// ---- POUs/Alle_Rum/Gange/Gang_5_153A/Visualization_4_330_1_1.TcVIS
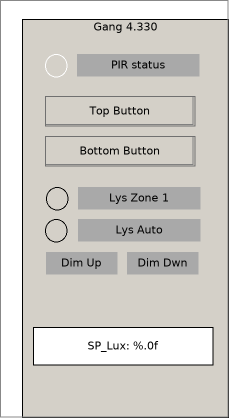
VISUALIZATION Visualization_4_330_1_1  // 229x418
    RoundedRectangle (22,19 207x399), "Gang 4.330"
    Rectangle (33,327 180x38), "SP_Lux: %.0f", text variable: P_Gang_5_135A.arrfbLysGruppe[1].fbLightCtrl.fLuxZone1
    Button (45,96 150x30), "Top Button"
        tap P_Gang_5_135A.bTopButtonZone1_Visu
    Button (45,136 150x30), "Bottom Button"
        tap P_Gang_5_135A.bBottomButtonZone1_Visu
    Ellipse (46,187 22x23), colour toggle: P_Gang_5_135A.fbLys.fbLightCtrl.bOnZone1
    Rectangle (78,187 122x22), "Lys Zone 1"
    Rectangle (46,252 71x22), "Dim Up", colour toggle: P_Gang_5_135A.arrfbLysGruppe[1].fbLightCtrl.bDimUp
    Rectangle (127,252 71x22), "Dim Dwn", colour toggle: P_Gang_5_135A.arrfbLysGruppe[1].fbLightCtrl.bDimDwn
    Ellipse (45,219 22x23), colour toggle: P_Gang_5_135A.arrfbLysGruppe[1].fbLightCtrl.bAutoZone1
    Rectangle (78,219 122x22), "Lys Auto"
    Ellipse (45,54 22x23), colour toggle: P_Gang_5_135A.arrfbLysGruppe[1].fbLightCtrl.bPIR
    Rectangle (77,54 122x22), "PIR status"
END_VISUALIZATION

// ---- POUs/Alle_Rum/Gange/Gang_5_149/Visualization_4_330_1_1_2.TcVIS
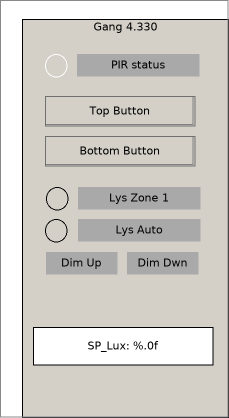
VISUALIZATION Visualization_4_330_1_1_2  // 229x418
    RoundedRectangle (22,19 207x399), "Gang 4.330"
    Rectangle (33,327 180x38), "SP_Lux: %.0f", text variable: P_Gang_5_135A.arrfbLysGruppe[1].fbLightCtrl.fLuxZone1
    Button (45,96 150x30), "Top Button"
        tap P_Gang_5_135A.bTopButtonZone1_Visu
    Button (45,136 150x30), "Bottom Button"
        tap P_Gang_5_135A.bBottomButtonZone1_Visu
    Ellipse (46,187 22x23), colour toggle: P_Gang_5_135A.fbLys.fbLightCtrl.bOnZone1
    Rectangle (78,187 122x22), "Lys Zone 1"
    Rectangle (46,252 71x22), "Dim Up", colour toggle: P_Gang_5_135A.arrfbLysGruppe[1].fbLightCtrl.bDimUp
    Rectangle (127,252 71x22), "Dim Dwn", colour toggle: P_Gang_5_135A.arrfbLysGruppe[1].fbLightCtrl.bDimDwn
    Ellipse (45,219 22x23), colour toggle: P_Gang_5_135A.arrfbLysGruppe[1].fbLightCtrl.bAutoZone1
    Rectangle (78,219 122x22), "Lys Auto"
    Ellipse (45,54 22x23), colour toggle: P_Gang_5_135A.arrfbLysGruppe[1].fbLightCtrl.bPIR
    Rectangle (77,54 122x22), "PIR status"
END_VISUALIZATION

// ---- POUs/Alle_Rum/Gange/Gang_7_119/Visualization_4_330_1_1_3.TcVIS
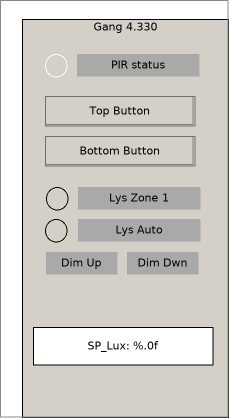
VISUALIZATION Visualization_4_330_1_1_3  // 229x418
    RoundedRectangle (22,19 207x399), "Gang 4.330"
    Rectangle (33,327 180x38), "SP_Lux: %.0f", text variable: P_Gang_5_135A.arrfbLysGruppe[1].fbLightCtrl.fLuxZone1
    Button (45,96 150x30), "Top Button"
        tap P_Gang_5_135A.bTopButtonZone1_Visu
    Button (45,136 150x30), "Bottom Button"
        tap P_Gang_5_135A.bBottomButtonZone1_Visu
    Ellipse (46,187 22x23), colour toggle: P_Gang_5_135A.fbLys.fbLightCtrl.bOnZone1
    Rectangle (78,187 122x22), "Lys Zone 1"
    Rectangle (46,252 71x22), "Dim Up", colour toggle: P_Gang_5_135A.arrfbLysGruppe[1].fbLightCtrl.bDimUp
    Rectangle (127,252 71x22), "Dim Dwn", colour toggle: P_Gang_5_135A.arrfbLysGruppe[1].fbLightCtrl.bDimDwn
    Ellipse (45,219 22x23), colour toggle: P_Gang_5_135A.arrfbLysGruppe[1].fbLightCtrl.bAutoZone1
    Rectangle (78,219 122x22), "Lys Auto"
    Ellipse (45,54 22x23), colour toggle: P_Gang_5_135A.arrfbLysGruppe[1].fbLightCtrl.bPIR
    Rectangle (77,54 122x22), "PIR status"
END_VISUALIZATION

// ---- POUs/Alle_Rum/Gange/Gang_5_153B/Visualization_4_330_1_1_1_1_1.TcVIS
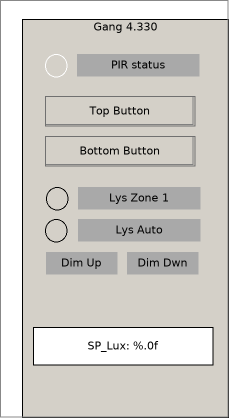
VISUALIZATION Visualization_4_330_1_1_1_1_1  // 229x418
    RoundedRectangle (22,19 207x399), "Gang 4.330"
    Rectangle (33,327 180x38), "SP_Lux: %.0f", text variable: P_Gang_5_135A.arrfbLysGruppe[1].fbLightCtrl.fLuxZone1
    Button (45,96 150x30), "Top Button"
        tap P_Gang_5_135A.bTopButtonZone1_Visu
    Button (45,136 150x30), "Bottom Button"
        tap P_Gang_5_135A.bBottomButtonZone1_Visu
    Ellipse (46,187 22x23), colour toggle: P_Gang_5_135A.fbLys.fbLightCtrl.bOnZone1
    Rectangle (78,187 122x22), "Lys Zone 1"
    Rectangle (46,252 71x22), "Dim Up", colour toggle: P_Gang_5_135A.arrfbLysGruppe[1].fbLightCtrl.bDimUp
    Rectangle (127,252 71x22), "Dim Dwn", colour toggle: P_Gang_5_135A.arrfbLysGruppe[1].fbLightCtrl.bDimDwn
    Ellipse (45,219 22x23), colour toggle: P_Gang_5_135A.arrfbLysGruppe[1].fbLightCtrl.bAutoZone1
    Rectangle (78,219 122x22), "Lys Auto"
    Ellipse (45,54 22x23), colour toggle: P_Gang_5_135A.arrfbLysGruppe[1].fbLightCtrl.bPIR
    Rectangle (77,54 122x22), "PIR status"
END_VISUALIZATION

// ---- POUs/Alle_Rum/Gange/Gang_5_145B/Visualization_4_330_1_1_1_1_1_1.TcVIS
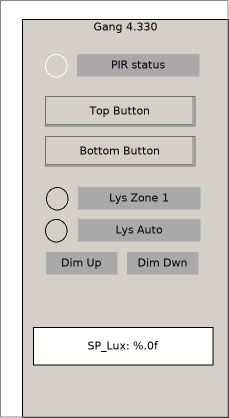
VISUALIZATION Visualization_4_330_1_1_1_1_1_1  // 229x418
    RoundedRectangle (22,19 207x399), "Gang 4.330"
    Rectangle (33,327 180x38), "SP_Lux: %.0f", text variable: P_Gang_5_135A.arrfbLysGruppe[1].fbLightCtrl.fLuxZone1
    Button (45,96 150x30), "Top Button"
        tap P_Gang_5_135A.bTopButtonZone1_Visu
    Button (45,136 150x30), "Bottom Button"
        tap P_Gang_5_135A.bBottomButtonZone1_Visu
    Ellipse (46,187 22x23), colour toggle: P_Gang_5_135A.fbLys.fbLightCtrl.bOnZone1
    Rectangle (78,187 122x22), "Lys Zone 1"
    Rectangle (46,252 71x22), "Dim Up", colour toggle: P_Gang_5_135A.arrfbLysGruppe[1].fbLightCtrl.bDimUp
    Rectangle (127,252 71x22), "Dim Dwn", colour toggle: P_Gang_5_135A.arrfbLysGruppe[1].fbLightCtrl.bDimDwn
    Ellipse (45,219 22x23), colour toggle: P_Gang_5_135A.arrfbLysGruppe[1].fbLightCtrl.bAutoZone1
    Rectangle (78,219 122x22), "Lys Auto"
    Ellipse (45,54 22x23), colour toggle: P_Gang_5_135A.arrfbLysGruppe[1].fbLightCtrl.bPIR
    Rectangle (77,54 122x22), "PIR status"
END_VISUALIZATION

// ---- POUs/Alle_Rum/Gange/Gang_5_153D/Visualization_4_330_1_1_1.TcVIS
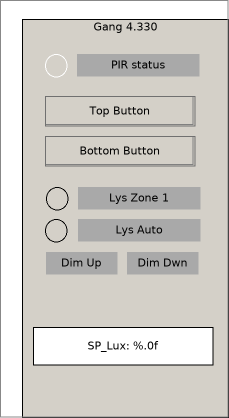
VISUALIZATION Visualization_4_330_1_1_1  // 229x418
    RoundedRectangle (22,19 207x399), "Gang 4.330"
    Rectangle (33,327 180x38), "SP_Lux: %.0f", text variable: P_Gang_5_135A.arrfbLysGruppe[1].fbLightCtrl.fLuxZone1
    Button (45,96 150x30), "Top Button"
        tap P_Gang_5_135A.bTopButtonZone1_Visu
    Button (45,136 150x30), "Bottom Button"
        tap P_Gang_5_135A.bBottomButtonZone1_Visu
    Ellipse (46,187 22x23), colour toggle: P_Gang_5_135A.fbLys.fbLightCtrl.bOnZone1
    Rectangle (78,187 122x22), "Lys Zone 1"
    Rectangle (46,252 71x22), "Dim Up", colour toggle: P_Gang_5_135A.arrfbLysGruppe[1].fbLightCtrl.bDimUp
    Rectangle (127,252 71x22), "Dim Dwn", colour toggle: P_Gang_5_135A.arrfbLysGruppe[1].fbLightCtrl.bDimDwn
    Ellipse (45,219 22x23), colour toggle: P_Gang_5_135A.arrfbLysGruppe[1].fbLightCtrl.bAutoZone1
    Rectangle (78,219 122x22), "Lys Auto"
    Ellipse (45,54 22x23), colour toggle: P_Gang_5_135A.arrfbLysGruppe[1].fbLightCtrl.bPIR
    Rectangle (77,54 122x22), "PIR status"
END_VISUALIZATION

// ---- POUs/Alle_Rum/Gange/Gang_5_153C/Visualization_4_330_1_1_1_1.TcVIS
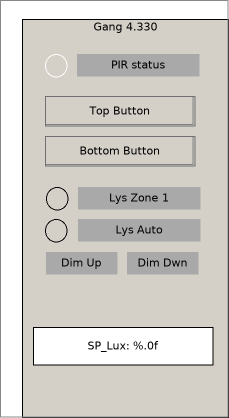
VISUALIZATION Visualization_4_330_1_1_1_1  // 229x418
    RoundedRectangle (22,19 207x399), "Gang 4.330"
    Rectangle (33,327 180x38), "SP_Lux: %.0f", text variable: P_Gang_5_135A.arrfbLysGruppe[1].fbLightCtrl.fLuxZone1
    Button (45,96 150x30), "Top Button"
        tap P_Gang_5_135A.bTopButtonZone1_Visu
    Button (45,136 150x30), "Bottom Button"
        tap P_Gang_5_135A.bBottomButtonZone1_Visu
    Ellipse (46,187 22x23), colour toggle: P_Gang_5_135A.fbLys.fbLightCtrl.bOnZone1
    Rectangle (78,187 122x22), "Lys Zone 1"
    Rectangle (46,252 71x22), "Dim Up", colour toggle: P_Gang_5_135A.arrfbLysGruppe[1].fbLightCtrl.bDimUp
    Rectangle (127,252 71x22), "Dim Dwn", colour toggle: P_Gang_5_135A.arrfbLysGruppe[1].fbLightCtrl.bDimDwn
    Ellipse (45,219 22x23), colour toggle: P_Gang_5_135A.arrfbLysGruppe[1].fbLightCtrl.bAutoZone1
    Rectangle (78,219 122x22), "Lys Auto"
    Ellipse (45,54 22x23), colour toggle: P_Gang_5_135A.arrfbLysGruppe[1].fbLightCtrl.bPIR
    Rectangle (77,54 122x22), "PIR status"
END_VISUALIZATION

// ---- POUs/Alle_Rum/Gange/Gang_x_xxx_2X2PCS_PIR_2LinjerLampe/Visualization_5_338.TcVIS
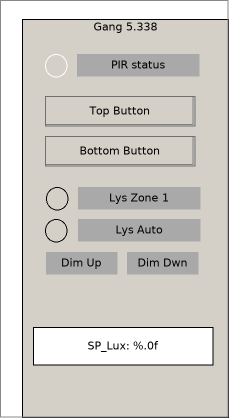
VISUALIZATION Visualization_5_338  // 229x418
    RoundedRectangle (22,19 207x399), "Gang 5.338"
    Rectangle (33,327 180x38), "SP_Lux: %.0f", text variable: P_Gang_5_338.arrfbLysGruppe[1].fbLightCtrl.fLuxZone1
    Button (45,96 150x30), "Top Button"
        tap P_Gang_5_338.bTopButtonZone1_Visu
    Button (45,136 150x30), "Bottom Button"
        tap P_Gang_5_338.bBottomButtonZone1_Visu
    Ellipse (46,187 22x23), colour toggle: P_Gang_5_338.arrfbLysGruppe[1].fbLightCtrl.bOnZone1
    Rectangle (78,187 122x22), "Lys Zone 1"
    Rectangle (46,252 71x22), "Dim Up", colour toggle: P_Gang_5_338.arrfbLysGruppe[1].fbLightCtrl.bDimUp
    Rectangle (127,252 71x22), "Dim Dwn", colour toggle: P_Gang_5_338.arrfbLysGruppe[1].fbLightCtrl.bDimDwn
    Ellipse (45,219 22x23), colour toggle: P_Gang_5_338.arrfbLysGruppe[1].fbLightCtrl.bAutoZone1
    Rectangle (78,219 122x22), "Lys Auto"
    Ellipse (45,54 22x23), colour toggle: P_Gang_5_338.arrfbLysGruppe[1].fbLightCtrl.bPIR
    Rectangle (77,54 122x22), "PIR status"
END_VISUALIZATION

// ---- POUs/Alle_Rum/Gange/Gang_5_146/Visualization_5_338_2.TcVIS
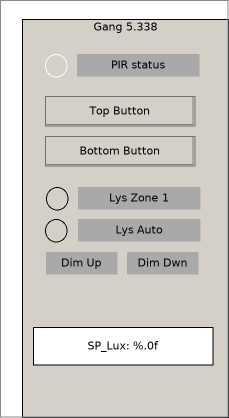
VISUALIZATION Visualization_5_338_2  // 229x418
    RoundedRectangle (22,19 207x399), "Gang 5.338"
    Rectangle (33,327 180x38), "SP_Lux: %.0f", text variable: P_Gang_5_338.arrfbLysGruppe[1].fbLightCtrl.fLuxZone1
    Button (45,96 150x30), "Top Button"
        tap P_Gang_5_338.bTopButtonZone1_Visu
    Button (45,136 150x30), "Bottom Button"
        tap P_Gang_5_338.bBottomButtonZone1_Visu
    Ellipse (46,187 22x23), colour toggle: P_Gang_5_338.arrfbLysGruppe[1].fbLightCtrl.bOnZone1
    Rectangle (78,187 122x22), "Lys Zone 1"
    Rectangle (46,252 71x22), "Dim Up", colour toggle: P_Gang_5_338.arrfbLysGruppe[1].fbLightCtrl.bDimUp
    Rectangle (127,252 71x22), "Dim Dwn", colour toggle: P_Gang_5_338.arrfbLysGruppe[1].fbLightCtrl.bDimDwn
    Ellipse (45,219 22x23), colour toggle: P_Gang_5_338.arrfbLysGruppe[1].fbLightCtrl.bAutoZone1
    Rectangle (78,219 122x22), "Lys Auto"
    Ellipse (45,54 22x23), colour toggle: P_Gang_5_338.arrfbLysGruppe[1].fbLightCtrl.bPIR
    Rectangle (77,54 122x22), "PIR status"
END_VISUALIZATION

// ---- POUs/Alle_Rum/Rum_Med_DALI_Pir/Rum_5_145A/Visualization_4_330_1_1_2_1.TcVIS
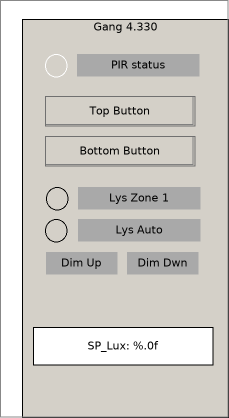
VISUALIZATION Visualization_4_330_1_1_2_1  // 229x418
    RoundedRectangle (22,19 207x399), "Gang 4.330"
    Rectangle (33,327 180x38), "SP_Lux: %.0f", text variable: P_Gang_5_135A.arrfbLysGruppe[1].fbLightCtrl.fLuxZone1
    Button (45,96 150x30), "Top Button"
        tap P_Gang_5_135A.bTopButtonZone1_Visu
    Button (45,136 150x30), "Bottom Button"
        tap P_Gang_5_135A.bBottomButtonZone1_Visu
    Ellipse (46,187 22x23), colour toggle: P_Gang_5_135A.fbLys.fbLightCtrl.bOnZone1
    Rectangle (78,187 122x22), "Lys Zone 1"
    Rectangle (46,252 71x22), "Dim Up", colour toggle: P_Gang_5_135A.arrfbLysGruppe[1].fbLightCtrl.bDimUp
    Rectangle (127,252 71x22), "Dim Dwn", colour toggle: P_Gang_5_135A.arrfbLysGruppe[1].fbLightCtrl.bDimDwn
    Ellipse (45,219 22x23), colour toggle: P_Gang_5_135A.arrfbLysGruppe[1].fbLightCtrl.bAutoZone1
    Rectangle (78,219 122x22), "Lys Auto"
    Ellipse (45,54 22x23), colour toggle: P_Gang_5_135A.arrfbLysGruppe[1].fbLightCtrl.bPIR
    Rectangle (77,54 122x22), "PIR status"
END_VISUALIZATION

// ---- POUs/Alle_Rum/Rum_Med_DALI_Pir/Rum_5_111B/Visualization_5_352_1_1_1_1_1.TcVIS
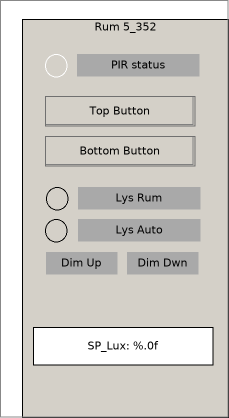
VISUALIZATION Visualization_5_352_1_1_1_1_1  // 229x418
    RoundedRectangle (22,19 207x399), "Rum 5_352"
    Rectangle (33,327 180x38), "SP_Lux: %.0f", text variable: P_Rum_4_324.fbLys.fbLightCtrl.fLuxZone1
    Button (45,96 150x30), "Top Button"
        tap P_Rum_5_352.bTopButtonZone1_Visu
    Button (45,136 150x30), "Bottom Button"
        tap P_Rum_5_352.bBottomButtonZone1_Visu
    Ellipse (46,187 22x23), colour toggle: P_Rum_5_352.fbLys.fbLightCtrl.bOnZone1
    Rectangle (78,187 122x22), "Lys Rum"
    Rectangle (46,252 71x22), "Dim Up", colour toggle: P_Rum_5_352.fbLys.fbLightCtrl.bDimUp
    Rectangle (127,252 71x22), "Dim Dwn", colour toggle: P_Rum_5_352.fbLys.fbLightCtrl.bDimDwn
    Ellipse (45,219 22x23), colour toggle: P_Rum_5_352.fbLys.fbLightCtrl.bAutoZone1
    Rectangle (78,219 122x22), "Lys Auto"
    Ellipse (45,54 22x23), colour toggle: P_Rum_5_352.fbLys.fbLightCtrl.bPIR
    Rectangle (77,54 122x22), "PIR status"
END_VISUALIZATION

// ---- POUs/DALI/DALI_Setup/VISUs/Visu_DALICommissioning.TcVIS
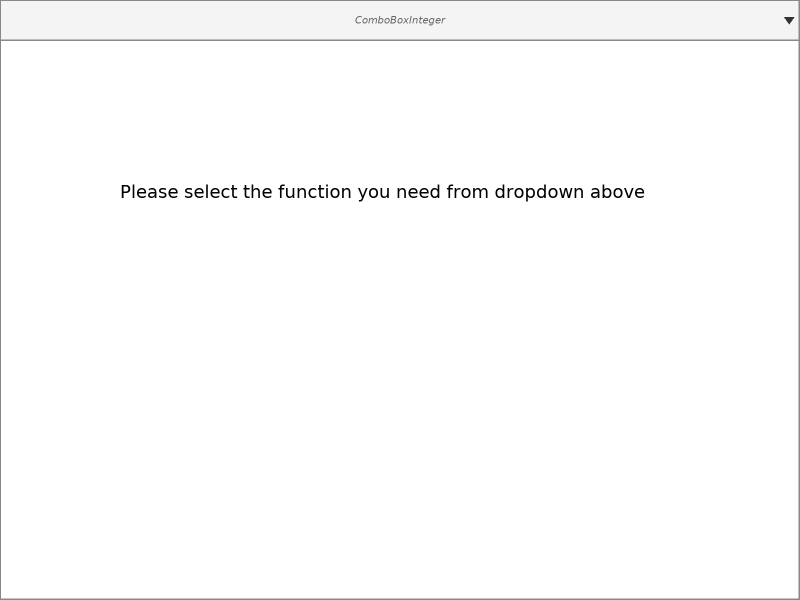
VISUALIZATION Visu_DALICommissioning  // 800x600
    ComboBoxInteger (0,0 800x40), variable: DALI_Commissioning.nSelectedDialog, input disabled if: DALI_Commissioning.bDisableComboBox, text list: 'TextList_Dialogs'
    Frame (0,40 800x560), frame switch variable: DALI_Commissioning.nSelectedDialog
        shows Visu_Welcome()
        shows Visu_Part102Commands()
        shows Visu_Part102Addressing()
        shows Visu_Part102Parameters()
        shows Visu_Part102Groups()
        shows Visu_Part102Scenes()
        shows Visu_Part102MemoryBank()
        shows Visu_Part102SetFading()
        shows Visu_Part202()
        shows Visu_Part205()
        shows Visu_Part207()
        shows Visu_Part208Switching()
        shows Visu_Part103Addressing()
        shows Visu_Part103Parameters()
        shows Visu_Part103Identify()
        shows Visu_Part301PushButton()
        shows Visu_Part302AbsoluteInputDevice()
        shows Visu_Part303OccupancySensor()
        shows Visu_Part304LightSensor()
        shows Visu_Part300GenericDevice()
        shows Visu_Part103MemoryBank()
        shows Visu_KL6821Configuration()
END_VISUALIZATION

// ---- POUs/DALI/DALI_Setup/VISUs/Visu_DALICommissioning/Visu_Part103Identify.TcVIS
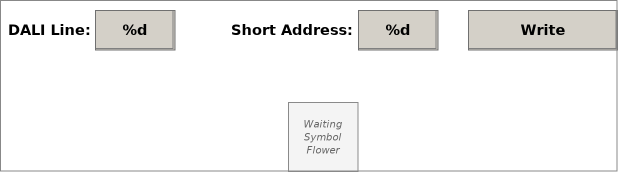
VISUALIZATION Visu_Part103Identify  // 618x172
    Button (468,10 150x40), "Write"
        OnMouseClick: execute { DALI_Commissioning.fbPart103IdentifyDevice.bWrite := TRUE; }
    WaitingSymbolFlower (288,102 70x70), invisible if: DALI_Commissioning.fbPart103MemoryPages.bHideWaitSymbol
    Textfield (228,10 130x40), "Short Address:"
    Button (358,10 80x40), "%d", text variable: DALI_Commissioning.fbPart103IdentifyDevice.nAddress
        OnMouseClick: write the text variable via Default, min 0, max 63, title "Insert Short Address"
    Group (5,10 170x40)
        Textfield (0,0 110x40), "DALI Line:"
        Button (90,0 80x40), "%d", text variable: GVL_Internal.nDALILine
            OnMouseClick: write the text variable via Default, min 1, max 10, title "Choose line"
END_VISUALIZATION

// ---- POUs/DALI/DALI_Setup/VISUs/Visu_DALICommissioning/Visu_Part208Switching.TcVIS
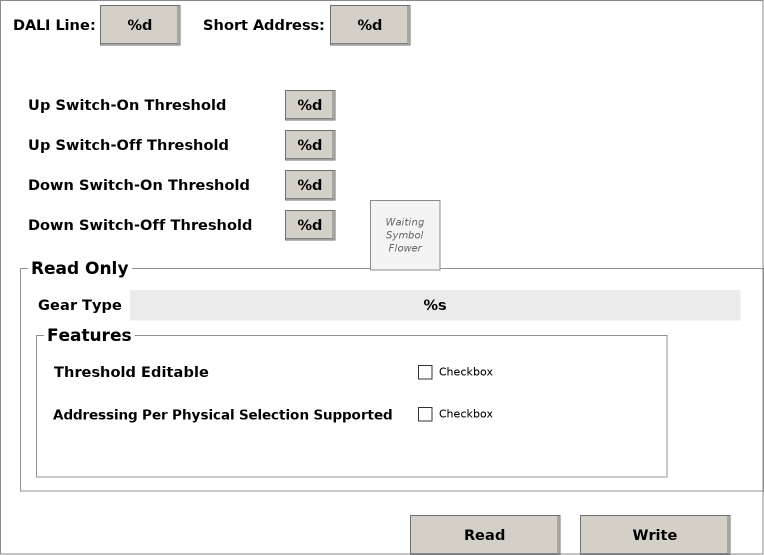
VISUALIZATION Visu_Part208Switching  // 764x555
    Group (200,5 210x40)
        Textfield (0,0 130x40), "Short Address:"
        Button (130,0 80x40), "%d", text variable: DALI_Commissioning.fbPart208Switching.nAddress
            OnMouseClick: write the text variable via Default, min 0, max 63, title "Insert Short Address"
    Group (10,5 170x40)
        Textfield (0,0 110x40), "DALI Line:"
        Button (90,0 80x40), "%d", text variable: GVL_Internal.nDALILine
            OnMouseClick: write the text variable via Default, min 1, max 10, title "Choose line"
    Textfield (25,90 250x30), "Up Switch-On Threshold"
    Textfield (25,130 250x30), "Up Switch-Off Threshold"
    Textfield (25,170 250x30), "Down Switch-On Threshold"
    Textfield (25,210 250x30), "Down Switch-Off Threshold"
    GroupBox (20,260 744x231), "Read Only"
        Textfield (15,30 250x30), "Gear Type"
        Textfield (110,30 610x30), "%s", text variable: DALI_Commissioning.fbPart208Switching.sGearType
        GroupBox (16,67 631x150), "Features"
            Checkbox (380,30 30x30), "Checkbox", variable: DALI_Commissioning.fbPart208Switching.bThreshold, input disabled if: TRUE
            Textfield (15,30 350x30), "Threshold Editable"
            Checkbox (380,72 30x30), "Checkbox", variable: DALI_Commissioning.fbPart208Switching.bAddressingPhysical, input disabled if: TRUE
    Textfield (50,400 355x30), "Addressing Per Physical Selection Supported"
    Button (410,515 150x40), "Read"
        OnMouseClick: execute { DALI_Commissioning.fbPart208Switching.bRead := TRUE; }
    Button (580,515 150x40), "Write"
        OnMouseClick: execute { DALI_Commissioning.fbPart208Switching.bWrite := TRUE; }
    WaitingSymbolFlower (370,200 70x70), invisible if: DALI_Commissioning.fbPart208Switching.bHideWaitSymbol
    Button (285,90 50x30), "%d", text variable: DALI_Commissioning.fbPart208Switching.nUpSwitchOnThreshold
        OnMouseClick: write the text variable via Default, min 0, max 255, title "Up Switch On Threshold"
    Button (285,130 50x30), "%d", text variable: DALI_Commissioning.fbPart208Switching.nUpSwitchOffThreshold
        OnMouseClick: write the text variable via Default, min 0, max 255, title "Up Switch Off Threshold"
    Button (285,170 50x30), "%d", text variable: DALI_Commissioning.fbPart208Switching.nDownSwitchOnThreshold
        OnMouseClick: write the text variable via Default, min 0, max 255, title "Down Switch On Threshold"
    Button (285,210 50x30), "%d", text variable: DALI_Commissioning.fbPart208Switching.nDownSwitchOffThreshold
        OnMouseClick: write the text variable via Default, min 0, max 255, title "Down Switch Off Threshold"
END_VISUALIZATION

// ---- POUs/DALI/DALI_Setup/VISUs/Visu_DALICommissioning/Visu_Welcome.TcVIS
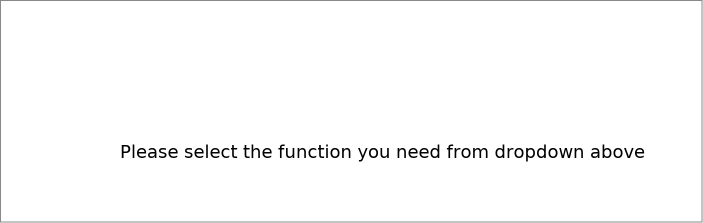
VISUALIZATION Visu_Welcome  // 703x223
    Rectangle (62,81 641x142), "Please select the function you need from dropdown above"
END_VISUALIZATION
